// TIA Portal project "DataProvider" (V14)

(* hardware
DEVICE "S7-1200 station_1"  S7-1200 Station
   slot 0: "Rack_0"  S7-1200 Rack  Rack  V1.0
   slot 1: "PLC_1"  CPU 1212C AC/DC/Rly  6ES7 212-1BE40-0XB0  V4.2
DEVICE "KP300BasicMono"  KP300 Basic mono PN
   slot 0: "KP300 Basic mono PN"  KP300 Basic mono PN  6AV6 647-0AH11-3AX0  12.0.0.0
   slot 1: "HMI_RT_1"  KP300 Basic mono PN  6AV6 647-0AH11-3AX0  12.0.0.0
   slot 5: "KP300BasicMono.IE_CP_1"  PROFINET Interface  12.0.0.0
      slot 1: "PROFINET Interface_1"  PROFINET Interface
         slot 1: "Eth0"  Port
*)

// ===== PLC "PLC_1"  CPU 1212C AC/DC/Rly =====

VAR_GLOBAL   // PLC tag table "IOs_DefaultTable"
   "AI0" AT %IW64 : Int;
   "AI1" AT %IW66 : Int;
   "DO0" AT %Q0.0 : Bool;
   "DO1" AT %Q0.1 : Bool;
END_VAR

VAR_GLOBAL   // PLC tag table "Inputs_Converted_to_SI-Units"
   "AI0_Volts" AT %MD0 : Real;
   "AI1_Volts" AT %MD4 : Real;
   "AI0_TempCels" AT %MD16 : Real;
   "AI1_TempCels" AT %MD20 : Real;
END_VAR

VAR_GLOBAL   // PLC tag table "HMI_Interchange_Vars"
   "HMI_AI0_TempCels" AT %MD8 : Real;
   "HMI_AI1_TempCels" AT %MD12 : Real;
END_VAR

DATA_BLOCK "webHMIData"   // DB1
{ S7_Optimized_Access := 'TRUE' }
VERSION : 0.1
   VAR
      webHMI_AI0_TempCels : Real;
      webHMI_AI1_TempCels : Real;
      webHMI_DO0_User : Bool;
      webHMI_DO1_User : Bool;
      error_www : Int;
   END_VAR
BEGIN
END_DATA_BLOCK

ORGANIZATION_BLOCK "Main"   // OB1, SCL, ProgramCycle
TITLE = "Main Program Sweep (Cycle)"
{ S7_Optimized_Access := 'TRUE' }
VERSION : 0.1
   VAR_INPUT
      Initial_Call : Bool;   // Initial call of this OB
      Remanence : Bool;   // =True, if remanent data are available
   END_VAR
BEGIN
   // 0V => 0
   // 10V => 27648
   // 

   // Convert input to volts:
   "AI0_Volts" := INT_TO_REAL("AI0") / 27648 * 10;
   "AI1_Volts" := INT_TO_REAL("AI1") / 27648 * 10;

   // convert volts to temperature in degrees celsius
   "AI0_TempCels" := "AI0_Volts" * 250 / 5; // temperature module is not calibrated correctly
   "AI1_TempCels" := "AI1_Volts" * 250 / 5; // temperature module is not calibrated correctly

   // Copy tags to HMI tags
   "HMI_AI0_TempCels" := "AI0_TempCels";
   "HMI_AI1_TempCels" := "AI1_TempCels";
END_ORGANIZATION_BLOCK

ORGANIZATION_BLOCK "webHMI"   // OB123, SCL, ProgramCycle
TITLE = "Main Program Sweep (Cycle)"
{ S7_Optimized_Access := 'TRUE' }
VERSION : 0.1
   VAR_INPUT
      Initial_Call : Bool;   // Initial call of this OB
      Remanence : Bool;   // =True, if remanent data are available
   END_VAR
BEGIN
   // copy values to tags which were reserved for webHMI interaction
   "webHMIData".webHMI_AI0_TempCels := "AI0_TempCels";
   "webHMIData".webHMI_AI1_TempCels := "AI1_TempCels";

   // handle http requests
   "webHMIData".error_www := WWW("DB 333");

   // copy variables' content which can be set from webHMI
   "DO0" := "webHMIData".webHMI_DO0_User;
   "DO1" := "webHMIData".webHMI_DO1_User;
END_ORGANIZATION_BLOCK

(* ===== HMI "HMI_RT_1" =====
connection "HMI_Connection_1": ETHERNET, SMART_S7_1200_OMS

HMI tags "Default tag table"
   "HMI_AI0_TempCels" : Real = PLC HMI_AI0_TempCels AT %MD8, 1 s
   "HMI_AI1_TempCels" : Real = PLC HMI_AI1_TempCels AT %MD12, 1 s

screen "Screen_1" 240x80
   IOField "I/O field_1" at 56,3 size 90x23; FormatPattern s999999999.999
      ProcessValue <- "HMI_AI0_TempCels"
   TextField "Text field_1" at 2,3 size 49x15; Text '°C (AI 0):'
   TextField "Text field_2" at 2,23 size 49x15; Text '°C (AI 1):'
   IOField "I/O field_2" at 57,23 size 94x23; FormatPattern s999999999.999
      ProcessValue <- "HMI_AI1_TempCels"
*)